FUNCTION_BLOCK SM_Palletizer EXTENDS StateMachine
VAR_IN_OUT
	ioChainController : FB_ChainController;
END_VAR
VAR_OUTPUT
	
	bAllPartsPresent: BOOL;	
	
END_VAR
VAR

	fbDoneCycle : BoolOut;
	fbStepWorkerBusy : FB_StepWorker;
	
	scFirstFloor : SC_FirstFloor :=
	(
		sChainName := 'scFirstFloor',
		rChainController := ioChainController
	);
	
	scSecondFloor : SC_SecondFloor :=
	(
		sChainName := 'scSecondFloor',
		rChainController := ioChainController
	);
END_VAR

SUPER^();
scFirstFloor();
scSecondFloor();

bAllPartsPresent := scSecondFloor.bAllPartsPresent;
scSecondFloor.bPlateOpen := scFirstFloor.bPlateOpen;

METHOD PROTECTED   Busy : BOOL
VAR_INPUT
END_VAR
scFirstFloor(bExecute := TRUE);
scSecondFloor(bExecute := TRUE);
END_METHOD

METHOD PROTECTED  Error : BOOL
VAR_INPUT
END_VAR
END_METHOD

PROPERTY getDoneCycle : I_StepCondition
GET
getDoneCycle := fbDoneCycle;
END_GET
END_PROPERTY

METHOD PROTECTED  Idle : BOOL
VAR_INPUT
END_VAR
END_METHOD

METHOD PROTECTED  Init : BOOL
VAR_INPUT
END_VAR
ioChainController
	.addChain(itfChain := scFirstFloor)
	.addChain(itfChain := scSecondFloor);
	
Start();
END_METHOD

METHOD PROTECTED  Prepare : BOOL
VAR_INPUT
END_VAR
END_METHOD

METHOD PROTECTED  Ready : BOOL
VAR_INPUT
END_VAR
END_METHOD

METHOD PROTECTED  Waiting : BOOL
VAR_INPUT
END_VAR
END_METHOD

END_FUNCTION_BLOCK

(* stored: Version 1.1.0.1, ProductVersion 3.1.4024.2
   POU SM_Palletizer: Id {73a1f3d2-201c-42a5-94a2-081d42f8b358}, SpecialFunc None
   Method Busy: Id {d9e0814b-09a9-4c14-8872-e9e8a213db38}
   Method Error: Id {1e64e457-c3f7-4fa5-85b2-02fb48054177}
   Property getDoneCycle: Id {10630946-14f0-417b-8a72-9ea11d6f3ffa}
   Get Get: Id {81aca46c-aea3-436a-81f7-8d17ab991d2b}
   Method Idle: Id {c949880c-6009-49c1-9143-74a28d29b1c1}
   Method Init: Id {d70eb0e0-8e12-4f46-8c48-9d942d266afa}
   Method Prepare: Id {ee19a450-41b7-476e-aa8a-75b7d82d8dde}
   Method Ready: Id {42cd7ed1-7213-436f-b42d-812333345c3e}
   Method Waiting: Id {c788c4e8-167a-44b4-9b42-c1f47d88d166} *)
